INTERFACE I_ChunkedRequestsHeaderAccessor

METHOD PUBLIC TryGetChunkSequenceFromRequest : BOOL
VAR_INPUT
	Request : I_Request;
	Destination : REFERENCE TO DINT;
END_VAR
END_METHOD

METHOD PUBLIC TryGetChunkTotalFromRequest : BOOL
VAR_INPUT
	Request : I_Request;
	Destination : REFERENCE TO DINT;
END_VAR
END_METHOD

METHOD PUBLIC TryGetHasMoreChunksFromRequest : BOOL
VAR_INPUT
	Request : I_Request;
	Destination : REFERENCE TO BOOL;
END_VAR
END_METHOD

METHOD PUBLIC TryGetRequestIdFromRequest : BOOL
VAR_INPUT
	Request : I_Request;
	Destination : REFERENCE TO T_MAXSTRING;
END_VAR
END_METHOD

METHOD PUBLIC TryGetSessionIdFromRequest : BOOL
VAR_INPUT
	Request : I_Request;
	Destination : REFERENCE TO T_MAXSTRING;
END_VAR
END_METHOD

END_INTERFACE

(* stored: Version 1.1.0.1, ProductVersion 3.1.4024.12
   Itf I_ChunkedRequestsHeaderAccessor: Id {cdf74b0f-d21f-4451-b9ee-85eec7aa413a}
   Method TryGetChunkSequenceFromRequest: Id {11f1b26f-e484-4358-9de5-2bcf4e4f6510}
   Method TryGetChunkTotalFromRequest: Id {26891607-e6a2-4757-a772-1ce94b7e2530}
   Method TryGetHasMoreChunksFromRequest: Id {4ee825c9-9bd4-4603-a4eb-2f1dcd13740b}
   Method TryGetRequestIdFromRequest: Id {23112332-f1af-4201-9485-5ad8f8ebf422}
   Method TryGetSessionIdFromRequest: Id {1efe8051-9e37-4188-bb4b-f0704a92e750} *)
